(* Logix 5000 project; controller EIP_Test2 1769-L16ER-BB1B rev 21.11; software revision 21.00 *)

TASK MainTask (continuous, watchdog 500 ms) : MainProgram

MODULES
   Local : 1769-L16ER-BB1B (PointIO 0, rev 21.11)
      T2 : vendor 1316 type 43 code 256 (Ethernet 192.168.4.6, rev 2.86, StandardDataDriven RPI 10 ms)
      Laser : vendor 1316 type 43 code 256 (Ethernet 192.168.4.3, rev 2.86, StandardDataDriven RPI 10 ms)
      Discrete_IO : Embedded (PointIO 1, rev 21.11, Output RPI 20 ms)
END_MODULES

TYPE Job_Field :
STRUCT
   Field_Index : SINT;
   Uniqueness : SINT;
   Verify : SINT;
   Reserved : SINT;
END_STRUCT
END_TYPE

TYPE LEC_O2T :
STRUCT
   X_Offset_mm_x100 : INT;   // X axis offset in units of [millimeters times 100]
   Y_Offset_mm_x100 : INT;   // Y axis offset in units of [millimeters times 100]
   Rotation_deg_x10 : INT;   // Rotation in units of [degrees times 10]
   X_Rotation_Center_mm_x100 : INT;   // X coordinate of the center of rotation in units of [millimeters times 100]
   Y_Rotation_Center_mm_x100 : INT;   // Y coordinate of the center of rotation in units of [millimeters times 100]
   X_Scale_x1000 : INT;   // X scale factor in units of [scale times 1000]. For example, use 1000 for a scale of 1
   Y_Scale_x1000 : INT;   // Y scale factor in units of [scale times 1000]. For example, use 1000 for a scale of 1
   Reserved : INT;   // Reserved
   Marker_Command : INT;   // Numeric command from PLC to marker
   Computed_Job_Field_Index : INT;   // The field index number for the computed field
   Mark_Timeout_Sec : INT;   // The maximum time to allow for marking [seconds]. An error is generated if this time is exceeded.
   Reserved_1 : INT;   // Reserved
   Barcode_Pass_Grade : INT;   // Pass grade for barcode verification
   Max_Remarks : INT;   // Maximum number of remark attempts if camera verification fails
   Short_Job_Field : Job_Field[5];   // The field index numbers of up to five 32-character string fields
   Long_Job_Field : Job_Field;   // The field index numbers of a single 64-character string field
   Marker_Job_File_Name : String32;   // The name of the marker job file to load
   Camera_Job_File_Name : String32;   // The name of the camera job file to load
   Short_Field_String : String32[5];   // Short string field values [32-characters]
   Long_Field_String : String128;   // Long string field value [128-characters]
END_STRUCT
END_TYPE

TYPE LEC_T2O :
STRUCT
   Marker_State : INT;   // The numeric marker state
   Reserved : INT;
   Last_Mark_Cycle_Time_Ms : DINT;   // The elapsed cycle time, or cycle time of the last mark in milliseconds
   Status_Word : DINT;   // LEC Standard IO word
   Marker_Error_Code : INT;   // The marker error code (0 = No Error)
   Controller_Error_Code : INT;   // The controller error code (LEC or Couth) (0 = No Error)
   Heart_Beat : DINT;   // Heartbeat indicator. Increasing number.
   Input_Field_Checksum : DINT;   // Simple checksum of all input field bytes
   Echo_Job_File_Name : String32;   // An echo of the job file name that has been loaded
   Results_Field : String128;   // A string results field generated by the marker
   Marker_State_Desc : String64;   // A description of the current marker state
   Marker_Error_Desc : String128;   // A description of the current marker error
END_STRUCT
END_TYPE

TYPE MDrive_Inputs_T2O :
STRUCT
   BY : BOOL;
   MV : BOOL;
   IN : SINT;
   C1 : DINT;
   C2 : DINT;
   V : DINT;
END_STRUCT
END_TYPE

TYPE MDrive_Outputs_O2T :
STRUCT
   A : DINT;
   D : DINT;
   MA : DINT;
   MR : DINT;
   RC : SINT;
   HC : SINT;
   OT : SINT;
   SL : DINT;
   VI : DINT;
   VM : DINT;
   TE : SINT;
   D5 : SINT;
END_STRUCT
END_TYPE

TYPE String128 :
STRUCT
   LEN : DINT;
   DATA : SINT[128];
END_STRUCT
END_TYPE

TYPE String32 :
STRUCT
   LEN : DINT;
   DATA : SINT[32];
END_STRUCT
END_TYPE

TYPE String64 :
STRUCT
   LEN : DINT;
   DATA : SINT[64];
END_STRUCT
END_TYPE

ADD_ON_INSTRUCTION Acquire_Host_Mode   (* revision 1.0, vendor Mecco Marking & Traceability *)
VAR_IN_OUT
   Inputs : LEC_O2T; {required}
   Outputs : LEC_T2O; {required}
END_VAR
VAR_OUTPUT
   InProcess : BOOL; {access Read Only}
   Done : BOOL; {access Read Only}
END_VAR
VAR_IN_OUT
   nstate : DINT; {required}
END_VAR
VAR
   Comment : STRING; {access None}
END_VAR

ROUTINE Logic   (* ladder *)
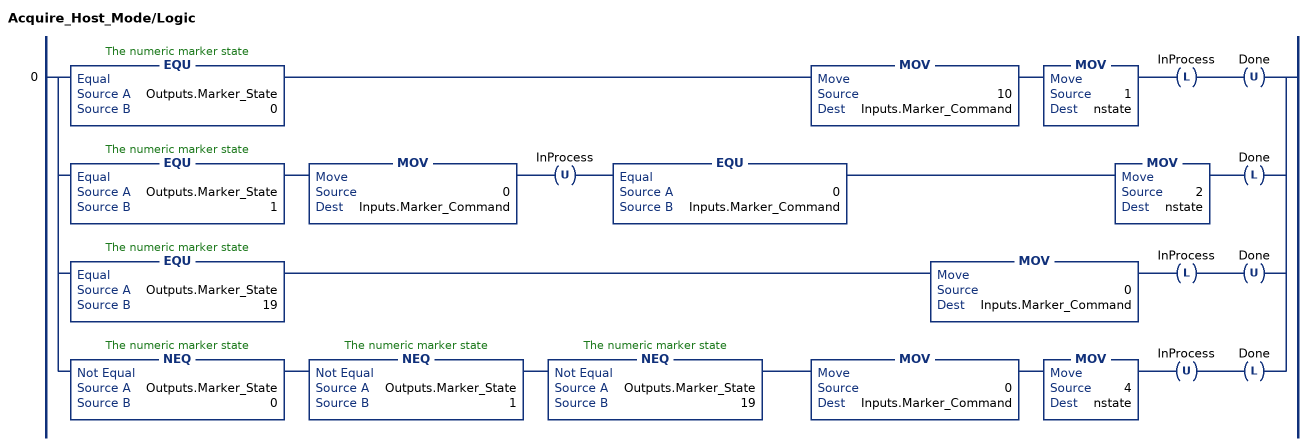
   0: [EQU(Outputs.Marker_State,0) MOV(10,Inputs.Marker_Command) MOV(1,nstate) OTL(InProcess) OTU(Done) ,EQU(Outputs.Marker_State,1) MOV(0,Inputs.Marker_Command) OTU(InProcess) EQU(0,Inputs.Marker_Command) MOV(2,nstate) OTL(Done) ,EQU(Outputs.Marker_State,19) MOV(0,Inputs.Marker_Command) OTL(InProcess) OTU(Done) ,NEQ(Outputs.Marker_State,0) NEQ(Outputs.Marker_State,1) NEQ(Outputs.Marker_State,19) MOV(0,Inputs.Marker_Command) MOV(4,nstate) OTU(InProcess) OTL(Done) ];
END_ROUTINE
END_ADD_ON_INSTRUCTION

ADD_ON_INSTRUCTION Clear_Error   (* revision 0.6, vendor Mecco Marking & Traceability *)
VAR_IN_OUT
   Inputs : LEC_O2T; {required}
   Outputs : LEC_T2O; {required}
END_VAR
VAR_OUTPUT
   Outcome : DINT; {access Read Only}
   InProcess : BOOL; {access Read Only}
   Done : BOOL; {access Read Only}
END_VAR
VAR_IN_OUT
   nstate : DINT; {required}
END_VAR
VAR
   Comment : STRING; {access None}
END_VAR

ROUTINE Logic   (* ladder *)
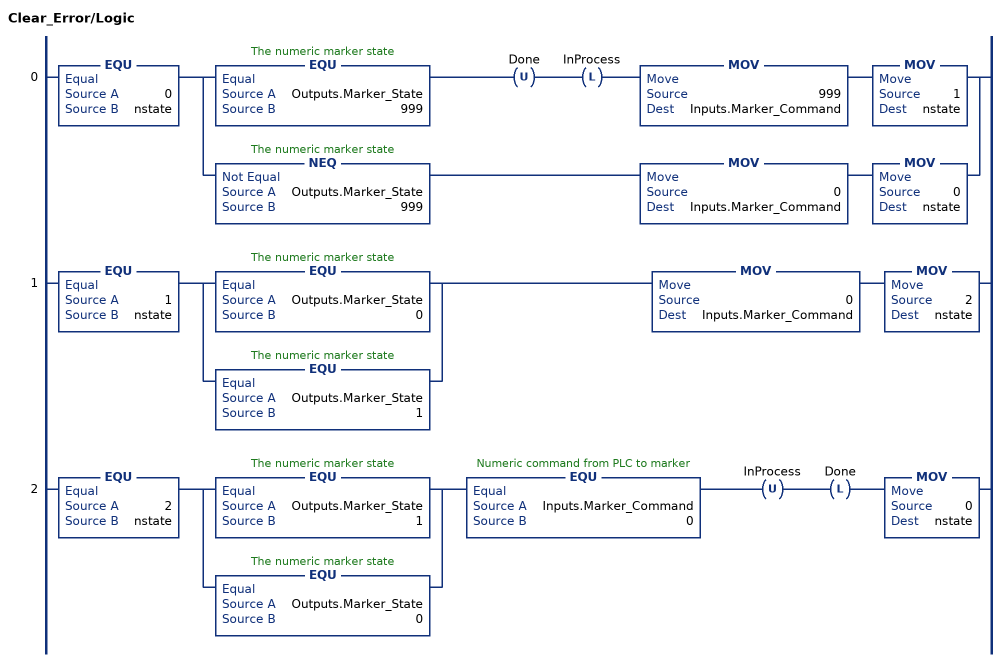
   0: EQU(0,nstate)[EQU(Outputs.Marker_State,999) OTU(Done) OTL(InProcess) MOV(999,Inputs.Marker_Command) MOV(1,nstate) ,NEQ(Outputs.Marker_State,999) MOV(0,Inputs.Marker_Command) MOV(0,nstate) ];
   1: EQU(1,nstate)[EQU(Outputs.Marker_State,0) ,EQU(Outputs.Marker_State,1) ]MOV(0,Inputs.Marker_Command)MOV(2,nstate);
   2: EQU(2,nstate)[EQU(Outputs.Marker_State,1) ,EQU(Outputs.Marker_State,0) ]EQU(Inputs.Marker_Command,0)OTU(InProcess)OTL(Done)MOV(0,nstate);
END_ROUTINE
END_ADD_ON_INSTRUCTION

ADD_ON_INSTRUCTION Load_Job   (* revision 1.0, vendor Mecco Marking & Traceability *)
VAR_IN_OUT
   Inputs : LEC_O2T; {required}
   Outputs : LEC_T2O; {required}
END_VAR
VAR_OUTPUT
   InProcess : BOOL; {access Read Only}
   Done : BOOL; {access Read Only}
END_VAR
VAR_IN_OUT
   Job_File_Name : STRING; {required}
END_VAR
VAR_OUTPUT
   Error : BOOL; {access Read Only}
END_VAR
VAR_INPUT
   Reset : BOOL;
END_VAR
VAR_IN_OUT
   nstate : DINT; {required}
END_VAR
VAR
   Comment : STRING; {access None}
   ErrorTimer : TIMER := (PRE := 5000); {access None}
   State1ONS : BOOL; {access None}
   BLANKSTRING : STRING; {access None}
   tnstate2 : TIMER := (PRE := 4000); {access None}
END_VAR

ROUTINE Logic   (* ladder *)
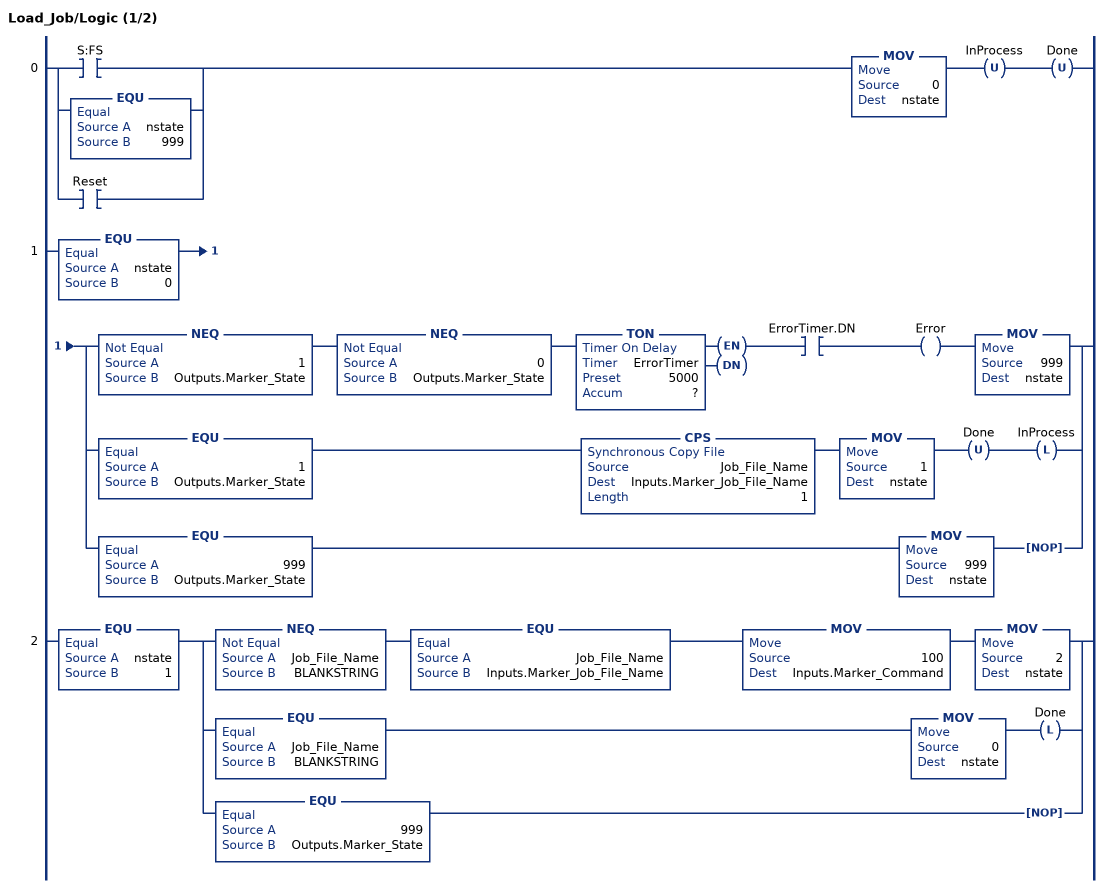
   0: [XIC(S:FS) ,EQU(nstate,999) ,XIC(Reset) ]MOV(0,nstate)OTU(InProcess)OTU(Done);
   1: EQU(nstate,0)[[NEQ(1,Outputs.Marker_State) NEQ(0,Outputs.Marker_State) TON(ErrorTimer,?,?) XIC(ErrorTimer.DN) OTE(Error) MOV(999,nstate) ,EQU(1,Outputs.Marker_State) CPS(Job_File_Name,Inputs.Marker_Job_File_Name,1) MOV(1,nstate) OTU(Done) OTL(InProcess) ] ,EQU(999,Outputs.Marker_State) MOV(999,nstate) NOP() ];
   2: EQU(nstate,1)[NEQ(Job_File_Name,BLANKSTRING) EQU(Job_File_Name,Inputs.Marker_Job_File_Name) MOV(100,Inputs.Marker_Command) MOV(2,nstate) ,EQU(Job_File_Name,BLANKSTRING) MOV(0,nstate) OTL(Done) ,EQU(999,Outputs.Marker_State) NOP() ];
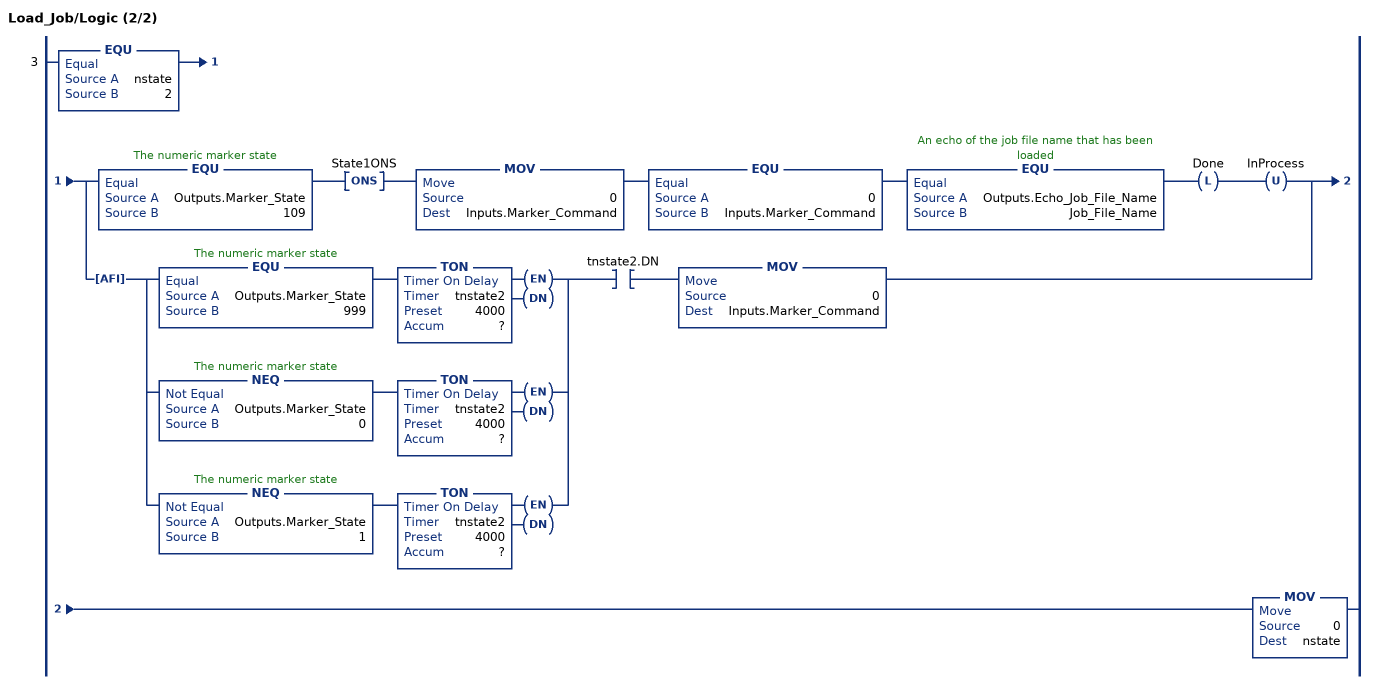
   3: EQU(nstate,2)[EQU(Outputs.Marker_State,109) ONS(State1ONS) MOV(0,Inputs.Marker_Command) EQU(0,Inputs.Marker_Command) EQU(Outputs.Echo_Job_File_Name,Job_File_Name) OTL(Done) OTU(InProcess) ,AFI() [EQU(Outputs.Marker_State,999) TON(tnstate2,?,?) ,NEQ(Outputs.Marker_State,0) TON(tnstate2,?,?) ,NEQ(Outputs.Marker_State,1) TON(tnstate2,?,?) ] XIC(tnstate2.DN) MOV(0,Inputs.Marker_Command) ]MOV(0,nstate);
END_ROUTINE
END_ADD_ON_INSTRUCTION

ADD_ON_INSTRUCTION Load_Job_T2   (* revision 1.0, vendor Mecco Marking & Traceability *)
VAR_IN_OUT
   Inputs : LEC_O2T; {required}
   Outputs : LEC_T2O; {required}
END_VAR
VAR_OUTPUT
   InProcess : BOOL; {access Read Only}
   Done : BOOL; {access Read Only}
END_VAR
VAR_IN_OUT
   Job_File_Name : STRING; {required}
END_VAR
VAR_OUTPUT
   Error : BOOL; {access Read Only}
END_VAR
VAR_INPUT
   Reset : BOOL;
END_VAR
VAR
   Comment : STRING; {access None}
   ErrorTimer : TIMER := (PRE := 5000); {access None}
   State1ONS : BOOL; {access None}
   BLANKSTRING : STRING; {access None}
   nstate : DINT; {access None}
END_VAR

ROUTINE Logic   (* ladder *)
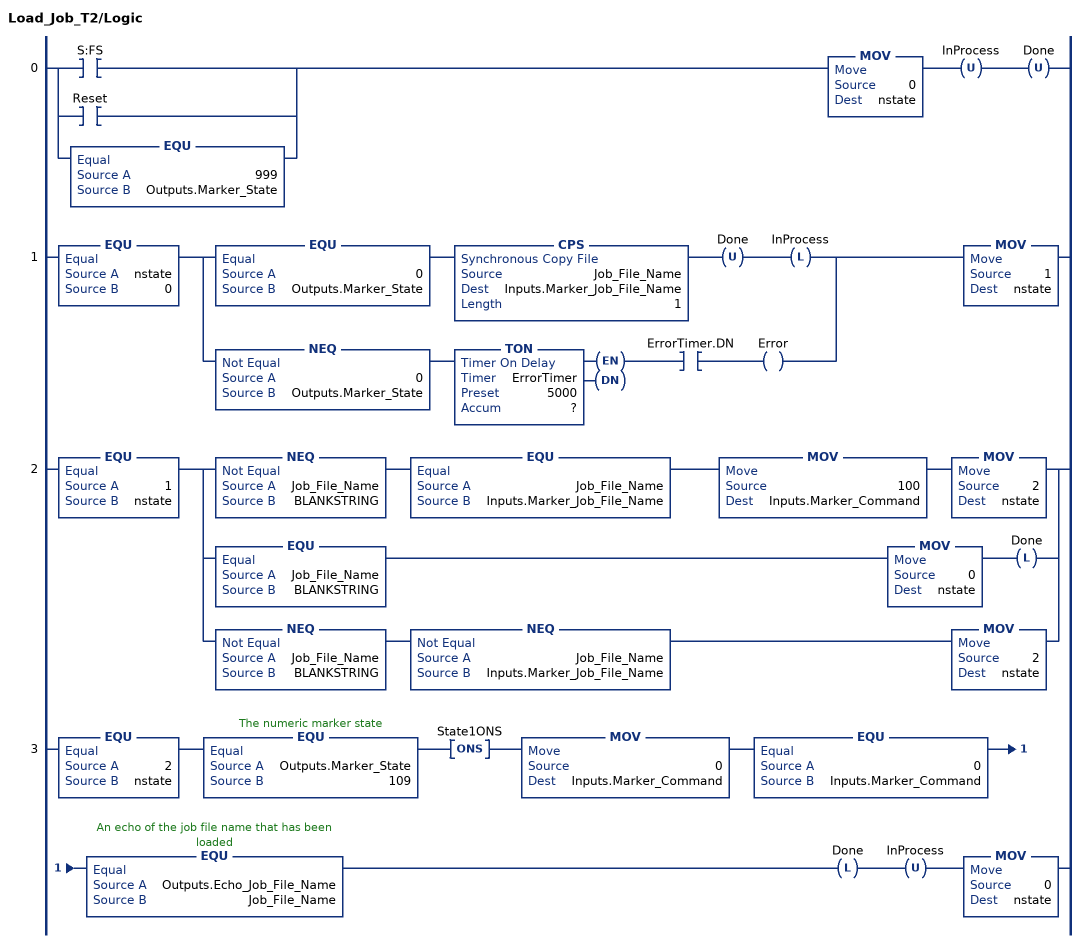
   0: [XIC(S:FS) ,XIC(Reset) ,EQU(999,Outputs.Marker_State) ]MOV(0,nstate)OTU(InProcess)OTU(Done);
   1: EQU(nstate,0)[EQU(0,Outputs.Marker_State) CPS(Job_File_Name,Inputs.Marker_Job_File_Name,1) OTU(Done) OTL(InProcess) ,NEQ(0,Outputs.Marker_State) TON(ErrorTimer,?,?) XIC(ErrorTimer.DN) OTE(Error) ]MOV(1,nstate);
   2: EQU(1,nstate)[NEQ(Job_File_Name,BLANKSTRING) EQU(Job_File_Name,Inputs.Marker_Job_File_Name) MOV(100,Inputs.Marker_Command) MOV(2,nstate) ,EQU(Job_File_Name,BLANKSTRING) MOV(0,nstate) OTL(Done) ,NEQ(Job_File_Name,BLANKSTRING) NEQ(Job_File_Name,Inputs.Marker_Job_File_Name) MOV(2,nstate) ];
   3: EQU(2,nstate)EQU(Outputs.Marker_State,109)ONS(State1ONS)MOV(0,Inputs.Marker_Command)EQU(0,Inputs.Marker_Command)EQU(Outputs.Echo_Job_File_Name,Job_File_Name)OTL(Done)OTU(InProcess)MOV(0,nstate);
END_ROUTINE
END_ADD_ON_INSTRUCTION

ADD_ON_INSTRUCTION Load_Variables   (* revision 1.0, vendor Mecco Marking & Traceability *)
VAR_IN_OUT
   Inputs : LEC_O2T; {required}
   Outputs : LEC_T2O; {required}
END_VAR
VAR_OUTPUT
   InProcess : BOOL; {access Read Only}
   Done : BOOL; {access Read Only}
END_VAR
VAR_IN_OUT
   Short_Variable_1_Text : STRING; {required}
END_VAR
VAR_INPUT
   Short_Variable_1_ObjectNum : DINT; {access None}
END_VAR
VAR_IN_OUT
   Short_Variable_2_Text : STRING; {required}
END_VAR
VAR_INPUT
   Short_Variable_2_ObjectNum : DINT; {access None}
END_VAR
VAR_IN_OUT
   Short_Variable_3_Text : STRING; {required}
END_VAR
VAR_INPUT
   Short_Variable_3_ObjectNum : DINT; {access None}
END_VAR
VAR_IN_OUT
   Short_Variable_4_Text : STRING; {required}
END_VAR
VAR_INPUT
   Short_Variable_4_ObjectNum : DINT; {access None}
END_VAR
VAR_IN_OUT
   Short_Variable_5_Text : STRING; {required}
END_VAR
VAR_INPUT
   Short_Variable_5_ObjectNum : DINT; {access None}
END_VAR
VAR_IN_OUT
   Long_Variable_Text : STRING; {required}
END_VAR
VAR_INPUT
   Long_Variable_ObjectNum : DINT; {access None}
END_VAR
VAR
   Comment : STRING; {access None}
   nstate : DINT := 3; {access None}
END_VAR

ROUTINE Logic   (* ladder *)
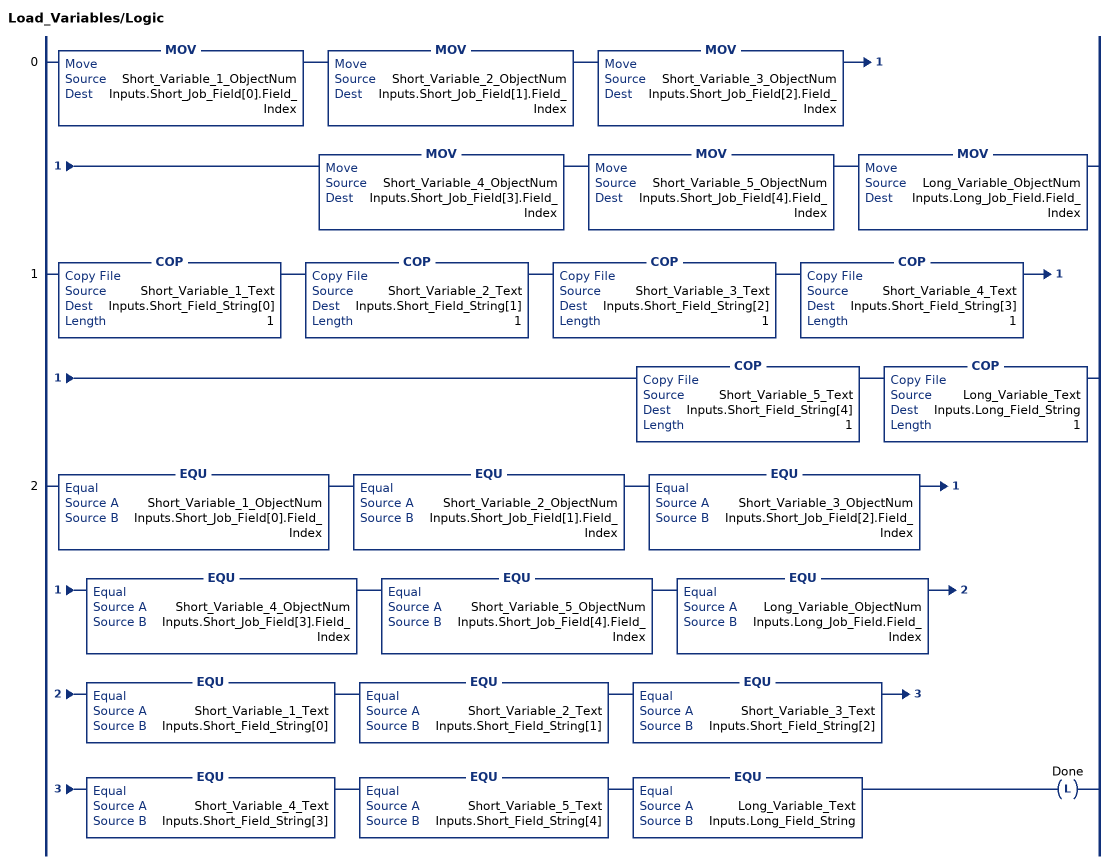
   0: MOV(Short_Variable_1_ObjectNum,Inputs.Short_Job_Field[0].Field_Index)MOV(Short_Variable_2_ObjectNum,Inputs.Short_Job_Field[1].Field_Index)MOV(Short_Variable_3_ObjectNum,Inputs.Short_Job_Field[2].Field_Index)MOV(Short_Variable_4_ObjectNum,Inputs.Short_Job_Field[3].Field_Index)MOV(Short_Variable_5_ObjectNum,Inputs.Short_Job_Field[4].Field_Index)MOV(Long_Variable_ObjectNum,Inputs.Long_Job_Field.Field_Index);
   1: COP(Short_Variable_1_Text,Inputs.Short_Field_String[0],1)COP(Short_Variable_2_Text,Inputs.Short_Field_String[1],1)COP(Short_Variable_3_Text,Inputs.Short_Field_String[2],1)COP(Short_Variable_4_Text,Inputs.Short_Field_String[3],1)COP(Short_Variable_5_Text,Inputs.Short_Field_String[4],1)COP(Long_Variable_Text,Inputs.Long_Field_String,1);
   2: EQU(Short_Variable_1_ObjectNum,Inputs.Short_Job_Field[0].Field_Index)EQU(Short_Variable_2_ObjectNum,Inputs.Short_Job_Field[1].Field_Index)EQU(Short_Variable_3_ObjectNum,Inputs.Short_Job_Field[2].Field_Index)EQU(Short_Variable_4_ObjectNum,Inputs.Short_Job_Field[3].Field_Index)EQU(Short_Variable_5_ObjectNum,Inputs.Short_Job_Field[4].Field_Index)EQU(Long_Variable_ObjectNum,Inputs.Long_Job_Field.Field_Index)EQU(Short_Variable_1_Text,Inputs.Short_Field_String[0])EQU(Short_Variable_2_Text,Inputs.Short_Field_String[1])EQU(Short_Variable_3_Text,Inputs.Short_Field_String[2])EQU(Short_Variable_4_Text,Inputs.Short_Field_String[3])EQU(Short_Variable_5_Text,Inputs.Short_Field_String[4])EQU(Long_Variable_Text,Inputs.Long_Field_String)OTL(Done);
END_ROUTINE
END_ADD_ON_INSTRUCTION

ADD_ON_INSTRUCTION Mark_Job   (* revision 1.0, vendor Mecco Marking & Traceability *)
VAR_IN_OUT
   Inputs : LEC_O2T; {required}
   Outputs : LEC_T2O; {required}
END_VAR
VAR_OUTPUT
   InProcess : BOOL; {access Read Only}
   Done : BOOL; {access Read Only}
   Error : BOOL; {access Read Only}
   MarkInProgress : BOOL; {access Read Only, visible}
END_VAR
VAR_INPUT
   Reset : BOOL;
END_VAR
VAR_IN_OUT
   nstate : DINT; {required}
END_VAR
VAR
   Comment : STRING; {access None}
   ErrorTimer : TIMER := (PRE := 5000); {access None}
END_VAR

ROUTINE Logic   (* ladder *)
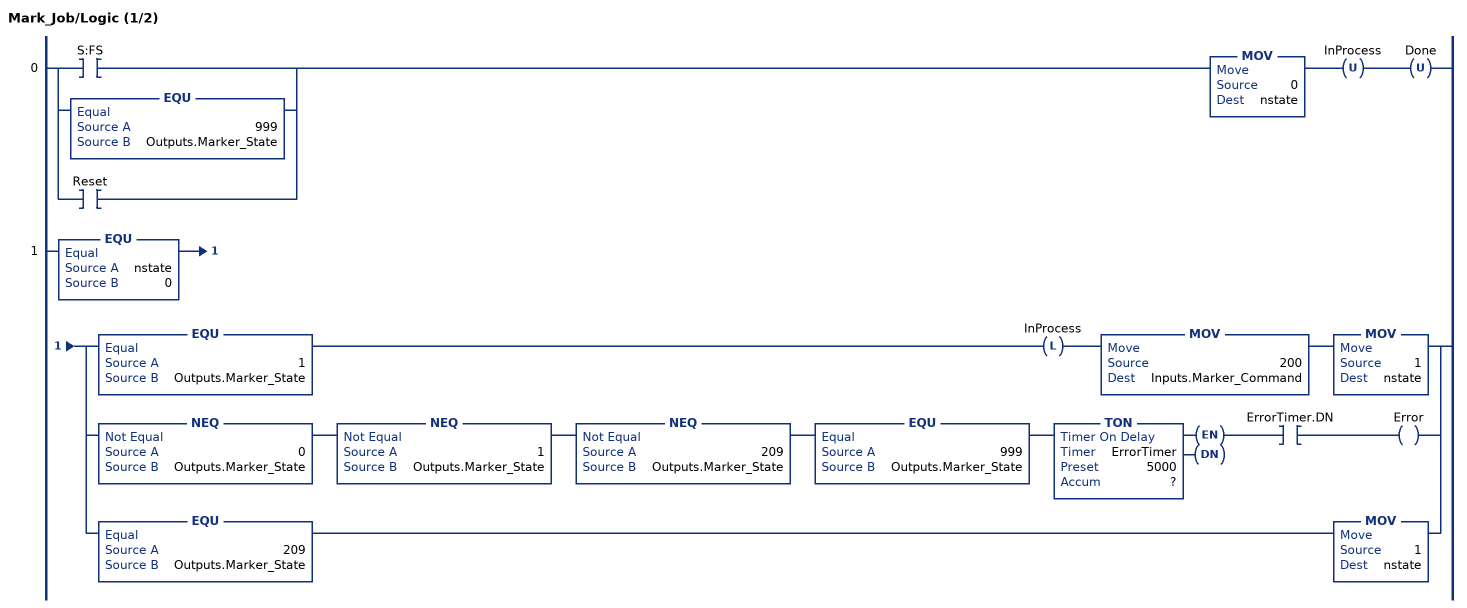
   0: [XIC(S:FS) ,EQU(999,Outputs.Marker_State) ,XIC(Reset) ]MOV(0,nstate)OTU(InProcess)OTU(Done);
   1: EQU(nstate,0)[EQU(1,Outputs.Marker_State) OTL(InProcess) MOV(200,Inputs.Marker_Command) MOV(1,nstate) ,NEQ(0,Outputs.Marker_State) NEQ(1,Outputs.Marker_State) NEQ(209,Outputs.Marker_State) EQU(999,Outputs.Marker_State) TON(ErrorTimer,?,?) XIC(ErrorTimer.DN) OTE(Error) ,EQU(209,Outputs.Marker_State) MOV(1,nstate) ];
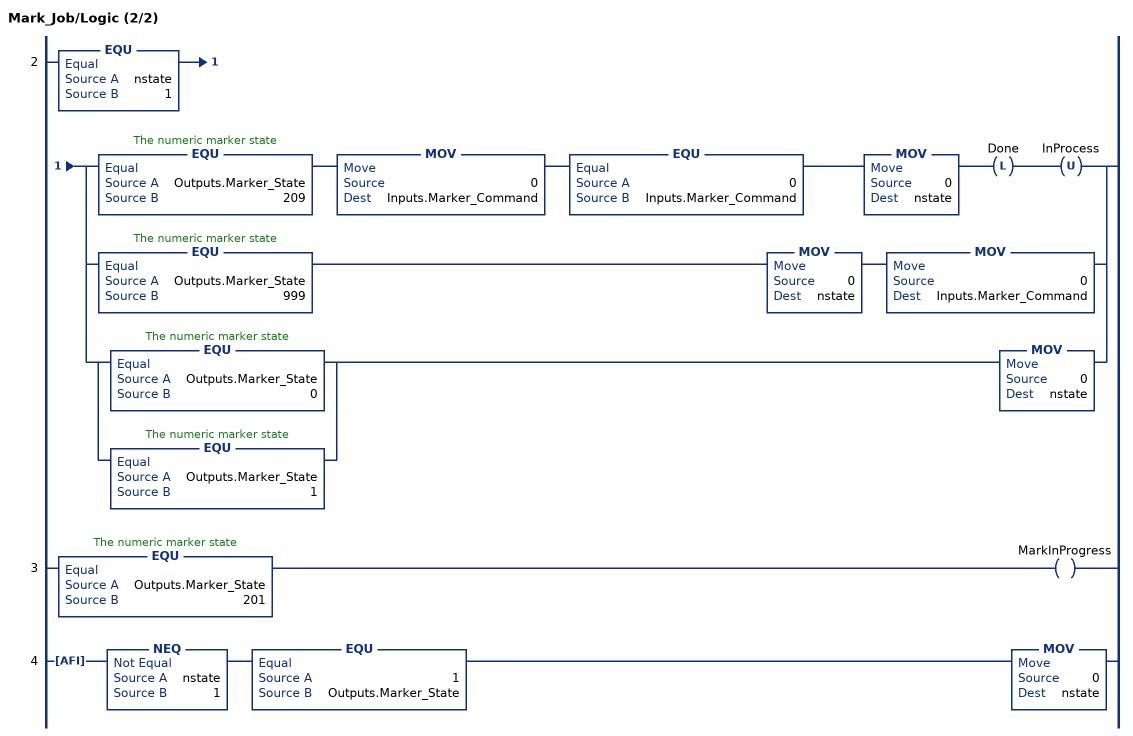
   2: EQU(nstate,1)[EQU(Outputs.Marker_State,209) MOV(0,Inputs.Marker_Command) EQU(0,Inputs.Marker_Command) MOV(0,nstate) OTL(Done) OTU(InProcess) ,EQU(Outputs.Marker_State,999) MOV(0,nstate) MOV(0,Inputs.Marker_Command) ,[EQU(Outputs.Marker_State,0) ,EQU(Outputs.Marker_State,1) ] MOV(0,nstate) ];
   3: EQU(Outputs.Marker_State,201)OTE(MarkInProgress);
   4: AFI()NEQ(nstate,1)EQU(1,Outputs.Marker_State)MOV(0,nstate);
END_ROUTINE
END_ADD_ON_INSTRUCTION

ADD_ON_INSTRUCTION Mark_Job_T2   (* revision 1.0, vendor Mecco Marking & Traceability *)
VAR_IN_OUT
   Inputs : LEC_O2T; {required}
   Outputs : LEC_T2O; {required}
END_VAR
VAR_OUTPUT
   InProcess : BOOL; {access Read Only}
   Done : BOOL; {access Read Only}
   Error : BOOL; {access Read Only}
   MarkInProgress : BOOL; {access Read Only, visible}
END_VAR
VAR_INPUT
   Reset : BOOL;
END_VAR
VAR
   Comment : STRING; {access None}
   ErrorTimer : TIMER := (PRE := 5000); {access None}
   nstate : DINT; {access None}
END_VAR

ROUTINE Logic   (* ladder *)
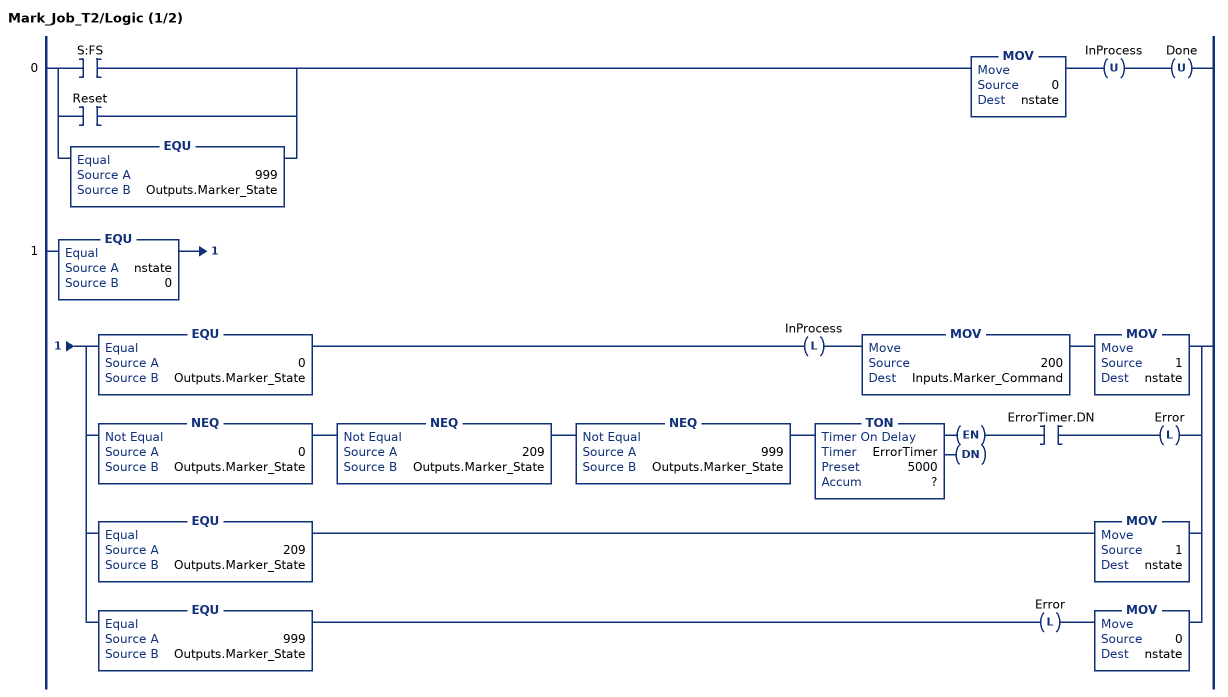
   0: [XIC(S:FS) ,[XIC(Reset) ,EQU(999,Outputs.Marker_State) ] ]MOV(0,nstate)OTU(InProcess)OTU(Done);
   1: EQU(nstate,0)[EQU(0,Outputs.Marker_State) OTL(InProcess) MOV(200,Inputs.Marker_Command) MOV(1,nstate) ,NEQ(0,Outputs.Marker_State) NEQ(209,Outputs.Marker_State) NEQ(999,Outputs.Marker_State) TON(ErrorTimer,?,?) XIC(ErrorTimer.DN) OTL(Error) ,EQU(209,Outputs.Marker_State) MOV(1,nstate) ,EQU(999,Outputs.Marker_State) OTL(Error) MOV(0,nstate) ];
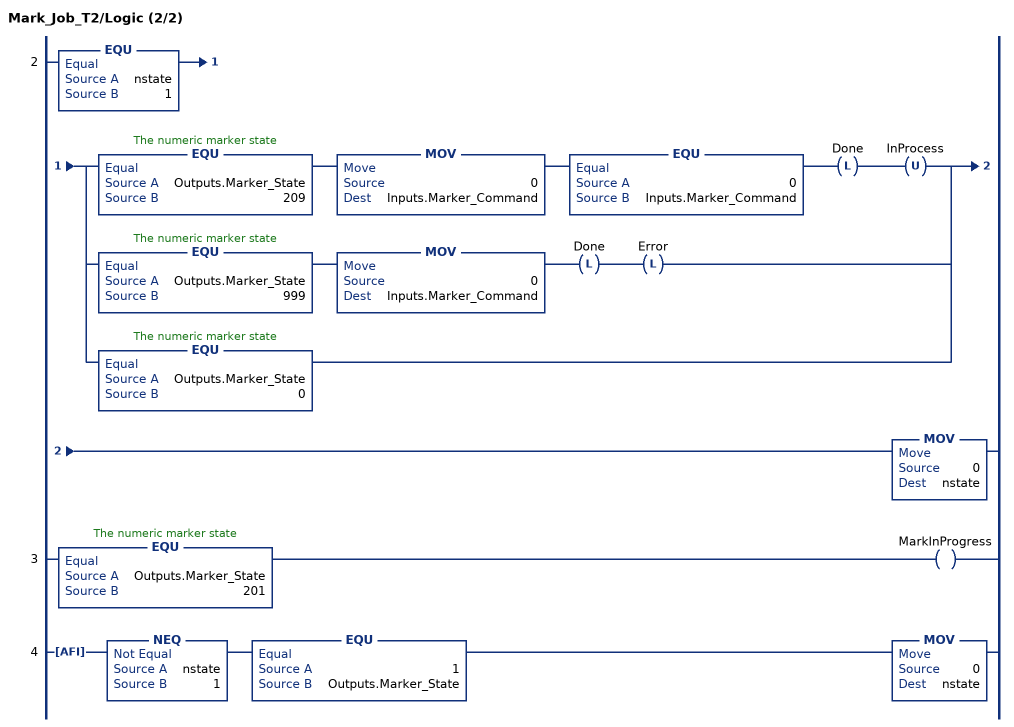
   2: EQU(nstate,1)[EQU(Outputs.Marker_State,209) MOV(0,Inputs.Marker_Command) EQU(0,Inputs.Marker_Command) OTL(Done) OTU(InProcess) ,EQU(Outputs.Marker_State,999) MOV(0,Inputs.Marker_Command) OTL(Done) OTL(Error) ,EQU(Outputs.Marker_State,0) ]MOV(0,nstate);
   3: EQU(Outputs.Marker_State,201)OTE(MarkInProgress);
   4: AFI()NEQ(nstate,1)EQU(1,Outputs.Marker_State)MOV(0,nstate);
END_ROUTINE
END_ADD_ON_INSTRUCTION

ADD_ON_INSTRUCTION Release_Host_Mode   (* revision 1.0, vendor Mecco Marking & Traceability *)
VAR_IN_OUT
   Inputs : LEC_O2T; {required}
   Outputs : LEC_T2O; {required}
END_VAR
VAR_OUTPUT
   InProcess : BOOL; {access Read Only}
   Done : BOOL; {access Read Only}
END_VAR
VAR
   Comment : STRING; {access None}
   nstate : DINT; {access None}
END_VAR

ROUTINE Logic   (* ladder *)
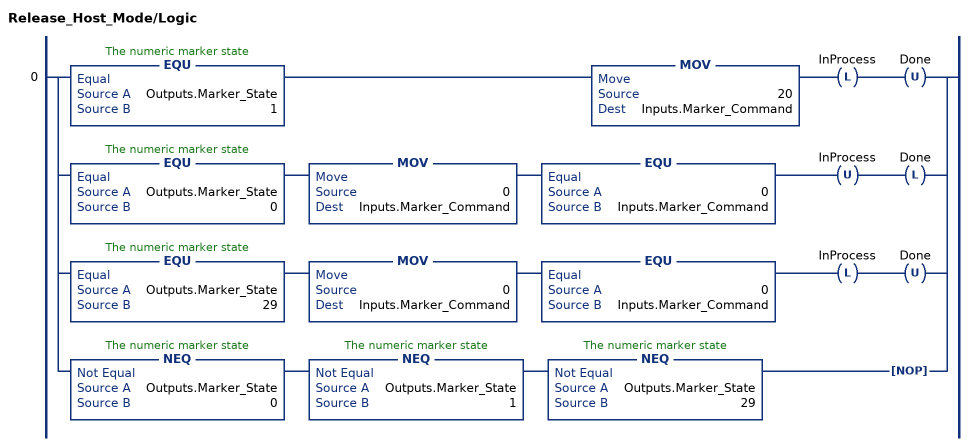
   0: [EQU(Outputs.Marker_State,1) MOV(20,Inputs.Marker_Command) OTL(InProcess) OTU(Done) ,EQU(Outputs.Marker_State,0) MOV(0,Inputs.Marker_Command) EQU(0,Inputs.Marker_Command) OTU(InProcess) OTL(Done) ,EQU(Outputs.Marker_State,29) MOV(0,Inputs.Marker_Command) EQU(0,Inputs.Marker_Command) OTL(InProcess) OTU(Done) ,NEQ(Outputs.Marker_State,0) NEQ(Outputs.Marker_State,1) NEQ(Outputs.Marker_State,29) NOP() ];
END_ROUTINE
END_ADD_ON_INSTRUCTION

VAR_GLOBAL   (* controller tags *)
   AcquireHost_nState : DINT;
   AOI_Acquire_Host_Laser : Acquire_Host_Mode;
   AOI_Load_Job : Load_Job;
   AOI_Load_Job_T2 : Load_Job_T2;
   AOI_Load_Variables : Load_Variables;
   AOI_Load_Variables_T2 : Load_Variables;
   AOI_Mark_Job : Mark_Job;
   AOI_Mark_Job_T2 : Mark_Job_T2;
   AOI_Release_Host : Release_Host_Mode;
   Dot_Peen_Input : LEC_O2T := (X_Scale_x1000 := 1000, Y_Scale_x1000 := 1000, Mark_Timeout_Sec := 999, Short_Job_Field[0].Field_Index := 1, Short_Job_Field[1].Field_Index := 2, Short_Job_Field[2].Field_Index := 3, Short_Job_Field[3].Field_Index := 4, Short_Job_Field[4].Field_Index := 5, Marker_Job_File_Name := 'Test1000.txt', Short_Field_String[0] := 'Line1', Short_Field_String[1] := 'Line2', Short_Field_String[2] := 'Line3', Short_Field_String[3] := 'Line4', Short_Field_String[4] := 'Line5');
   Dot_Peen_Load_Job : BOOL;
   Dot_Peen_Load_Variables : BOOL;
   Dot_Peen_Mark_Job : BOOL;
   Dot_Peen_Output : LEC_T2O := (Last_Mark_Cycle_Time_Ms := 4945, Heart_Beat := 345199, Input_Field_Checksum := 3222, Echo_Job_File_Name := 'Test1000.txt', Marker_State_Desc := '[1] Ready', Marker_Error_Desc := 'No error');
   HMI_Bits : DINT := 1;
   Job : BOOL;
   Laser_Acquire : BOOL;
   Laser_Acquire_Host : BOOL;
   Laser_Inputs : LEC_O2T := (X_Scale_x1000 := 1000, Y_Scale_x1000 := 1000, Mark_Timeout_Sec := 999, Short_Job_Field[0].Field_Index := 1, Short_Job_Field[1].Field_Index := 2, Short_Job_Field[2].Field_Index := 3, Short_Job_Field[3].Field_Index := 4, Short_Job_Field[4].Field_Index := 5, Marker_Job_File_Name := 'TAG1.DAT', Short_Field_String[0] := 'Line1', Short_Field_String[1] := 'Line2', Short_Field_String[2] := 'Line3', Short_Field_String[3] := 'Line4', Short_Field_String[4] := 'Line5', Long_Field_String := '590.00,3537,500,300,30,204.000,150,75,0,40.00,2.0,0,0,0,0,0.0,1,0,2.550,2.550,0.0,0.0,0,0');
   Laser_JobFileName : STRING;
   Laser_Load_Job : BOOL;
   Laser_Load_Variables : BOOL;
   Laser_Mark_Job : BOOL;
   Laser_Online_String : STRING := 'Ready to Fire';
   Laser_Outputs : LEC_T2O := (Marker_State := 1, Heart_Beat := 516904, Input_Field_Checksum := 7119, Echo_Job_File_Name := 'TAG1.DAT', Results_Field := '1405', Marker_State_Desc := '[1] Ready: Host Mode active', Marker_Error_Desc := 'No error');
   Laser_Release_Host : BOOL;
   LoadJob_nState : DINT;
   Long : STRING;
   Long_T2 : STRING;
   MarkJob_nState : DINT;
   MDive_Inputs : MDrive_Inputs_T2O;
   MDrive_Outputs : MDrive_Outputs_O2T;
   Short : STRING[5];
   Short_T2 : STRING[5];
   T2_JobFileName : STRING;
END_VAR

PROGRAM MainProgram   (* main routine MainRoutine *)
VAR
   B_Reset_Marker : BOOL;
   bDotPeenEnabled : BOOL := 1;
   Blank_String : String32;
   bLaserEnabled : BOOL := 1;
   bPauseDotPeen : BOOL;
   bPauseLaser : BOOL;
   Dot_Peen_Job_File_Name : String32 := 'Test1000.txt';
   Dot_Peen_Run_Counter : COUNTER := (ACC := 12, DN := 1);
   Dot_Peen_Start_Button : BOOL := 1;
   Field : String32[5] := ([0] := 'Line1', [1] := 'Line2', [2] := 'Line3', [3] := 'Line4', [4] := 'Line5');
   Job_File_Name : STRING := 'Series0_Text.dat';
   l_hstate : DINT;
   l_on : TIMER := (PRE := 12000);
   Laser_Heartbeat_Old : DINT := 1306452;
   Laser_Run_Counter : COUNTER := (ACC := 5, CU := 1, DN := 1);
   LASER_RUNNING : BOOL;
   LEC_Latch : BOOL;
   lHeartbeat_Check : BOOL := 1;
   lheartbeat_Timer : TIMER := (PRE := 1000);
   M_Drive_Accel_1 : BOOL;
   M_Drive_Decel_1 : BOOL;
   M_Drive_Position_1 : BOOL;
   M_Drive_Query_SN : BOOL;
   M_Drive_Reverse_1 : BOOL;
   M_Drive_Slew_1 : BOOL;
   M_Drive_Stop : BOOL;
   M_Drive_Velocity_1 : BOOL;
   MDrive_Out : DINT;
   nState : DINT;
   nState_DotPeen : DINT;
   Reset_Dot_Peen_Counter : BOOL;
   Reset_Laser_Counter : BOOL;
   Start_Button : BOOL := 1;
   T2_Latch : BOOL := 1;
   T_MarkerResetTimer : TIMER;
END_VAR

ROUTINE Dot_Peen   (* ladder *)
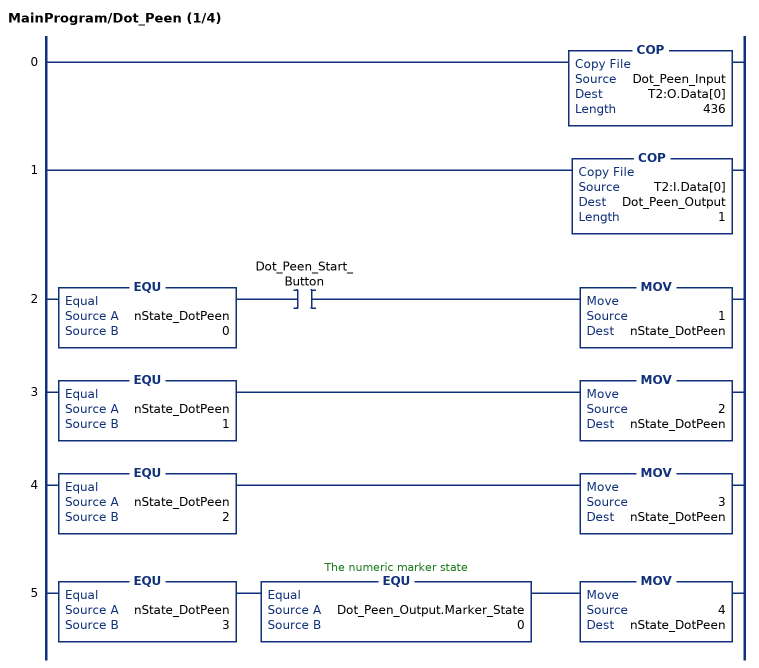
   0: COP(Dot_Peen_Input,T2:O.Data[0],436);
   1: COP(T2:I.Data[0],Dot_Peen_Output,1);
   2: EQU(nState_DotPeen,0)XIC(Dot_Peen_Start_Button)MOV(1,nState_DotPeen);
   3: EQU(nState_DotPeen,1)MOV(2,nState_DotPeen);
   4: EQU(nState_DotPeen,2)MOV(3,nState_DotPeen);
   5: EQU(nState_DotPeen,3)EQU(Dot_Peen_Output.Marker_State,0)MOV(4,nState_DotPeen);
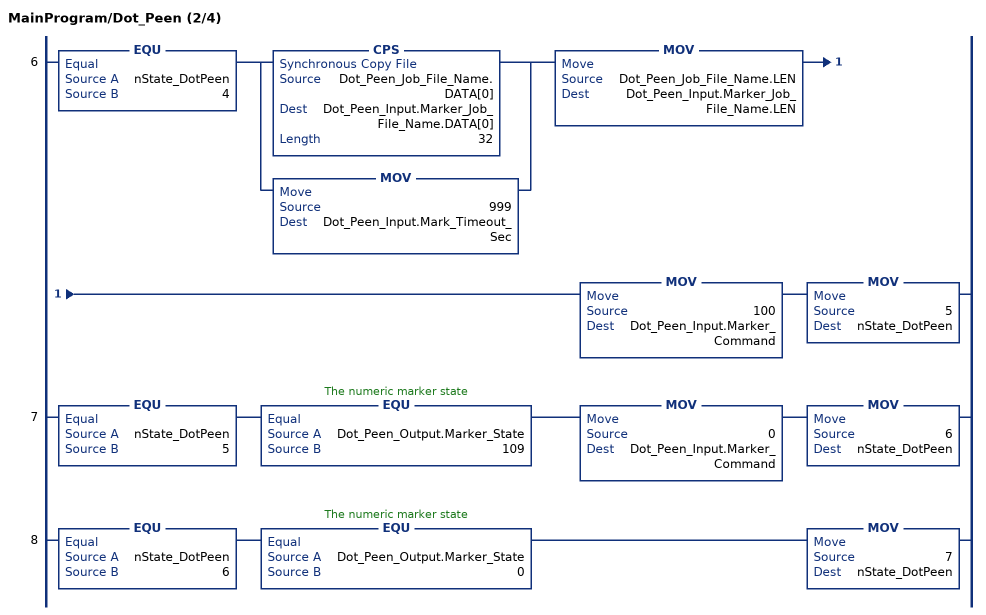
   6: EQU(nState_DotPeen,4)[CPS(Dot_Peen_Job_File_Name.DATA[0],Dot_Peen_Input.Marker_Job_File_Name.DATA[0],32) ,MOV(999,Dot_Peen_Input.Mark_Timeout_Sec) ]MOV(Dot_Peen_Job_File_Name.LEN,Dot_Peen_Input.Marker_Job_File_Name.LEN)MOV(100,Dot_Peen_Input.Marker_Command)MOV(5,nState_DotPeen);
   7: EQU(nState_DotPeen,5)EQU(Dot_Peen_Output.Marker_State,109)MOV(0,Dot_Peen_Input.Marker_Command)MOV(6,nState_DotPeen);
   8: EQU(nState_DotPeen,6)EQU(Dot_Peen_Output.Marker_State,0)MOV(7,nState_DotPeen);
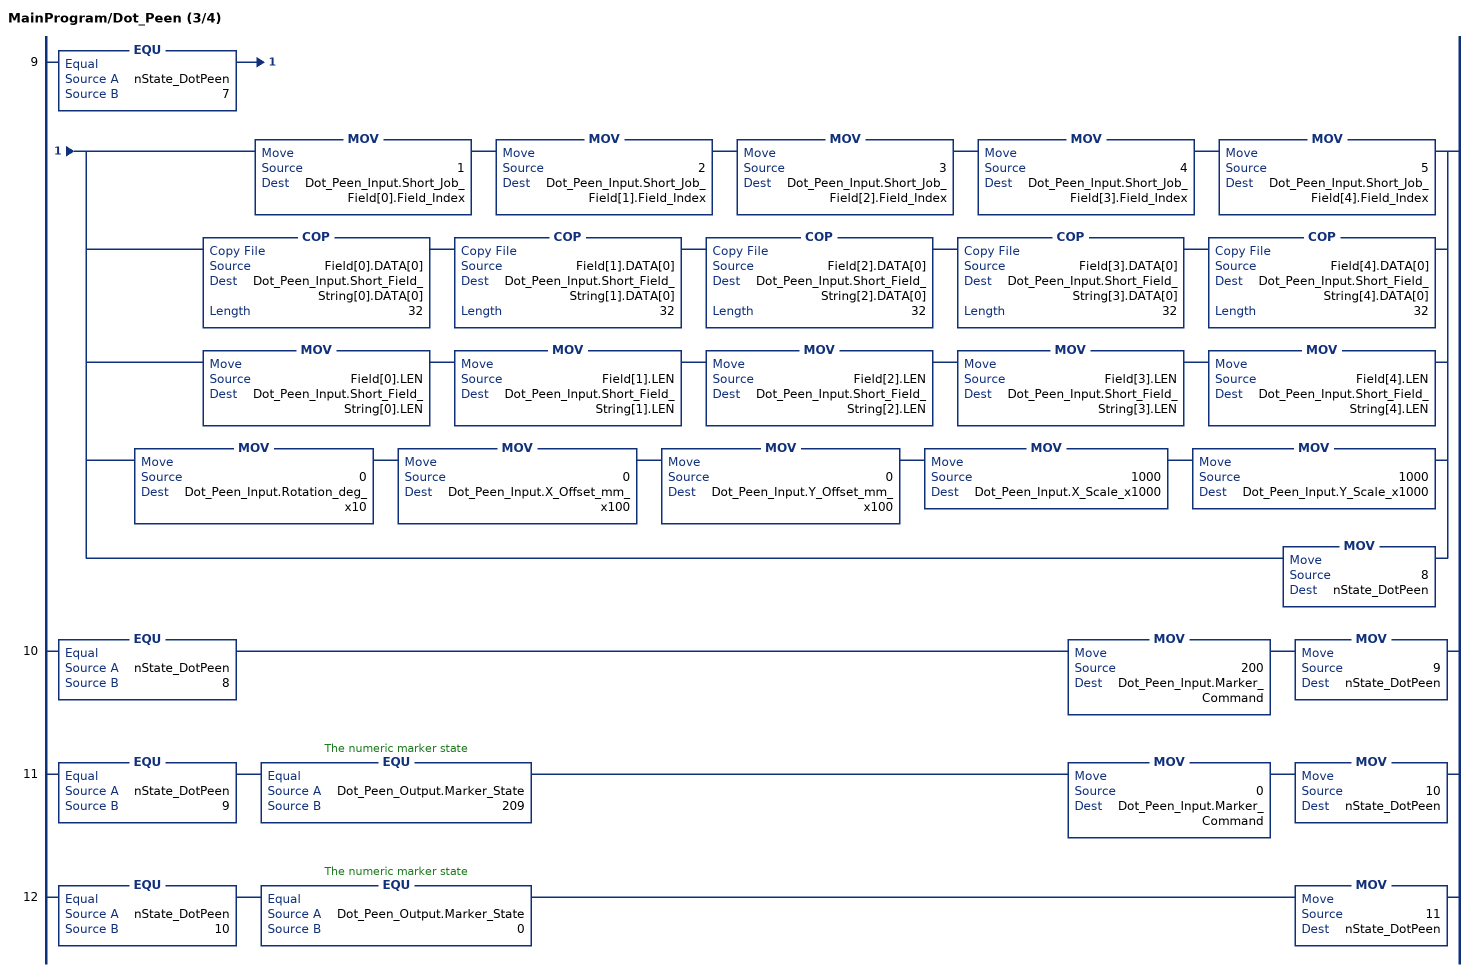
   9: EQU(nState_DotPeen,7)[MOV(1,Dot_Peen_Input.Short_Job_Field[0].Field_Index) MOV(2,Dot_Peen_Input.Short_Job_Field[1].Field_Index) MOV(3,Dot_Peen_Input.Short_Job_Field[2].Field_Index) MOV(4,Dot_Peen_Input.Short_Job_Field[3].Field_Index) MOV(5,Dot_Peen_Input.Short_Job_Field[4].Field_Index) ,COP(Field[0].DATA[0],Dot_Peen_Input.Short_Field_String[0].DATA[0],32) COP(Field[1].DATA[0],Dot_Peen_Input.Short_Field_String[1].DATA[0],32) COP(Field[2].DATA[0],Dot_Peen_Input.Short_Field_String[2].DATA[0],32) COP(Field[3].DATA[0],Dot_Peen_Input.Short_Field_String[3].DATA[0],32) COP(Field[4].DATA[0],Dot_Peen_Input.Short_Field_String[4].DATA[0],32) ,MOV(Field[0].LEN,Dot_Peen_Input.Short_Field_String[0].LEN) MOV(Field[1].LEN,Dot_Peen_Input.Short_Field_String[1].LEN) MOV(Field[2].LEN,Dot_Peen_Input.Short_Field_String[2].LEN) MOV(Field[3].LEN,Dot_Peen_Input.Short_Field_String[3].LEN) MOV(Field[4].LEN,Dot_Peen_Input.Short_Field_String[4].LEN) ,MOV(0,Dot_Peen_Input.Rotation_deg_x10) MOV(0,Dot_Peen_Input.X_Offset_mm_x100) MOV(0,Dot_Peen_Input.Y_Offset_mm_x100) MOV(1000,Dot_Peen_Input.X_Scale_x1000) MOV(1000,Dot_Peen_Input.Y_Scale_x1000) ,MOV(8,nState_DotPeen) ];
   10: EQU(nState_DotPeen,8)MOV(200,Dot_Peen_Input.Marker_Command)MOV(9,nState_DotPeen);
   11: EQU(nState_DotPeen,9)EQU(Dot_Peen_Output.Marker_State,209)MOV(0,Dot_Peen_Input.Marker_Command)MOV(10,nState_DotPeen);
   12: EQU(nState_DotPeen,10)EQU(Dot_Peen_Output.Marker_State,0)MOV(11,nState_DotPeen);
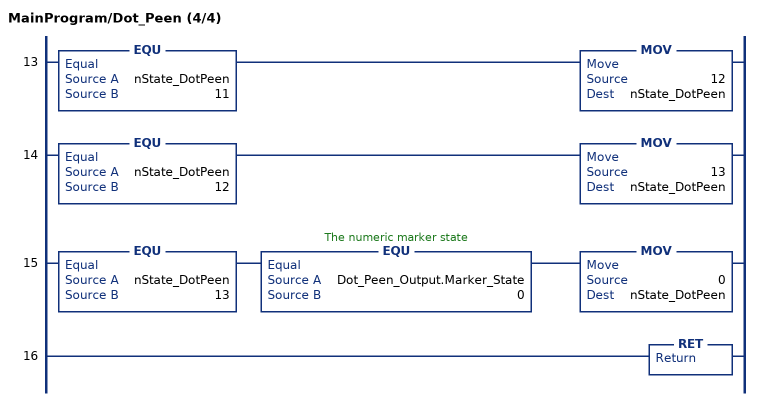
   13: EQU(nState_DotPeen,11)MOV(12,nState_DotPeen);
   14: EQU(nState_DotPeen,12)MOV(13,nState_DotPeen);
   15: EQU(nState_DotPeen,13)EQU(Dot_Peen_Output.Marker_State,0)MOV(0,nState_DotPeen);
   16: RET();
END_ROUTINE

ROUTINE Dot_Peen_AOI   (* ladder *)
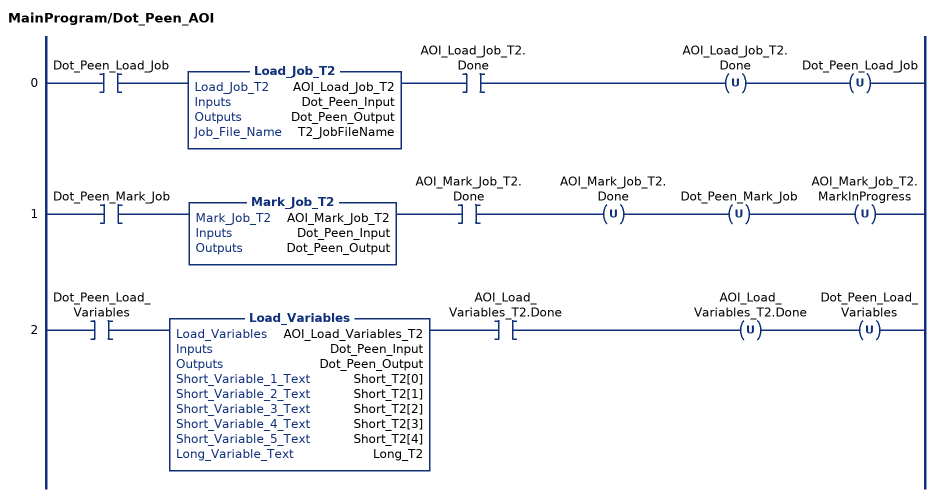
   0: XIC(Dot_Peen_Load_Job)Load_Job_T2(AOI_Load_Job_T2,Dot_Peen_Input,Dot_Peen_Output,T2_JobFileName)XIC(AOI_Load_Job_T2.Done)OTU(AOI_Load_Job_T2.Done)OTU(Dot_Peen_Load_Job);
   1: XIC(Dot_Peen_Mark_Job)Mark_Job_T2(AOI_Mark_Job_T2,Dot_Peen_Input,Dot_Peen_Output)XIC(AOI_Mark_Job_T2.Done)OTU(AOI_Mark_Job_T2.Done)OTU(Dot_Peen_Mark_Job)OTU(AOI_Mark_Job_T2.MarkInProgress);
   2: XIC(Dot_Peen_Load_Variables)Load_Variables(AOI_Load_Variables_T2,Dot_Peen_Input,Dot_Peen_Output,Short_T2[0],Short_T2[1],Short_T2[2],Short_T2[3],Short_T2[4],Long_T2)XIC(AOI_Load_Variables_T2.Done)OTU(AOI_Load_Variables_T2.Done)OTU(Dot_Peen_Load_Variables);
END_ROUTINE

ROUTINE Laser   (* ladder *)
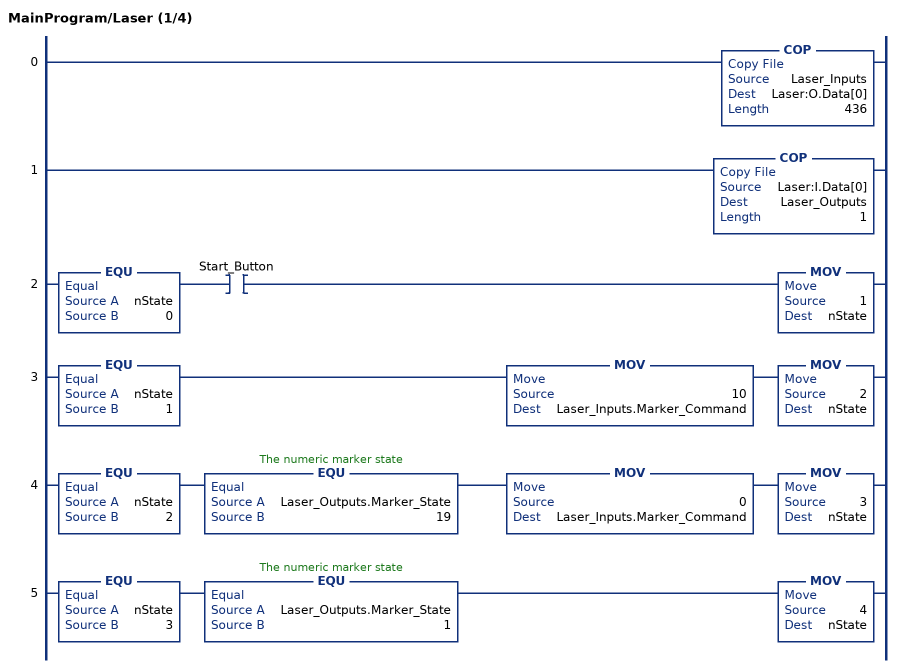
   0: COP(Laser_Inputs,Laser:O.Data[0],436);
   1: COP(Laser:I.Data[0],Laser_Outputs,1);
   2: EQU(nState,0)XIC(Start_Button)MOV(1,nState);
   3: EQU(nState,1)MOV(10,Laser_Inputs.Marker_Command)MOV(2,nState);
   4: EQU(nState,2)EQU(Laser_Outputs.Marker_State,19)MOV(0,Laser_Inputs.Marker_Command)MOV(3,nState);
   5: EQU(nState,3)EQU(Laser_Outputs.Marker_State,1)MOV(4,nState);
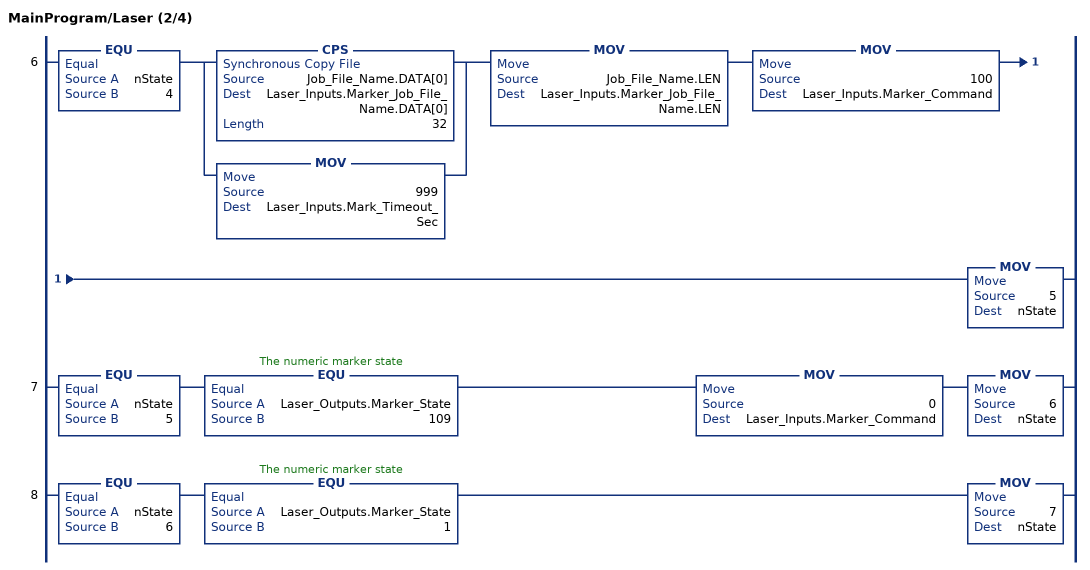
   6: EQU(nState,4)[CPS(Job_File_Name.DATA[0],Laser_Inputs.Marker_Job_File_Name.DATA[0],32) ,MOV(999,Laser_Inputs.Mark_Timeout_Sec) ]MOV(Job_File_Name.LEN,Laser_Inputs.Marker_Job_File_Name.LEN)MOV(100,Laser_Inputs.Marker_Command)MOV(5,nState);
   7: EQU(nState,5)EQU(Laser_Outputs.Marker_State,109)MOV(0,Laser_Inputs.Marker_Command)MOV(6,nState);
   8: EQU(nState,6)EQU(Laser_Outputs.Marker_State,1)MOV(7,nState);
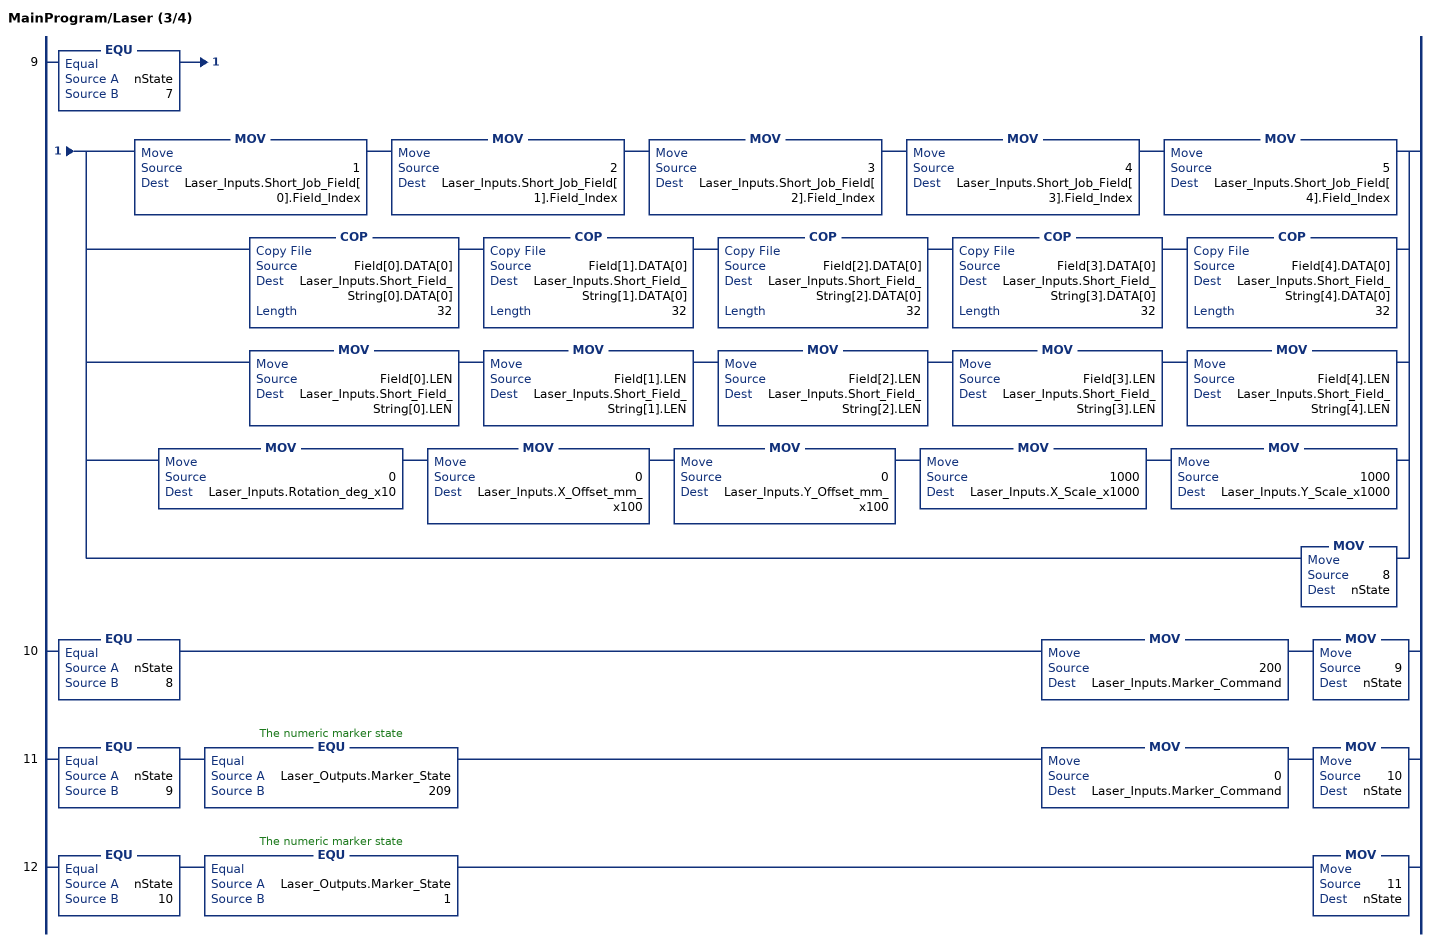
   9: EQU(nState,7)[MOV(1,Laser_Inputs.Short_Job_Field[0].Field_Index) MOV(2,Laser_Inputs.Short_Job_Field[1].Field_Index) MOV(3,Laser_Inputs.Short_Job_Field[2].Field_Index) MOV(4,Laser_Inputs.Short_Job_Field[3].Field_Index) MOV(5,Laser_Inputs.Short_Job_Field[4].Field_Index) ,COP(Field[0].DATA[0],Laser_Inputs.Short_Field_String[0].DATA[0],32) COP(Field[1].DATA[0],Laser_Inputs.Short_Field_String[1].DATA[0],32) COP(Field[2].DATA[0],Laser_Inputs.Short_Field_String[2].DATA[0],32) COP(Field[3].DATA[0],Laser_Inputs.Short_Field_String[3].DATA[0],32) COP(Field[4].DATA[0],Laser_Inputs.Short_Field_String[4].DATA[0],32) ,MOV(Field[0].LEN,Laser_Inputs.Short_Field_String[0].LEN) MOV(Field[1].LEN,Laser_Inputs.Short_Field_String[1].LEN) MOV(Field[2].LEN,Laser_Inputs.Short_Field_String[2].LEN) MOV(Field[3].LEN,Laser_Inputs.Short_Field_String[3].LEN) MOV(Field[4].LEN,Laser_Inputs.Short_Field_String[4].LEN) ,MOV(0,Laser_Inputs.Rotation_deg_x10) MOV(0,Laser_Inputs.X_Offset_mm_x100) MOV(0,Laser_Inputs.Y_Offset_mm_x100) MOV(1000,Laser_Inputs.X_Scale_x1000) MOV(1000,Laser_Inputs.Y_Scale_x1000) ,MOV(8,nState) ];
   10: EQU(nState,8)MOV(200,Laser_Inputs.Marker_Command)MOV(9,nState);
   11: EQU(nState,9)EQU(Laser_Outputs.Marker_State,209)MOV(0,Laser_Inputs.Marker_Command)MOV(10,nState);
   12: EQU(nState,10)EQU(Laser_Outputs.Marker_State,1)MOV(11,nState);
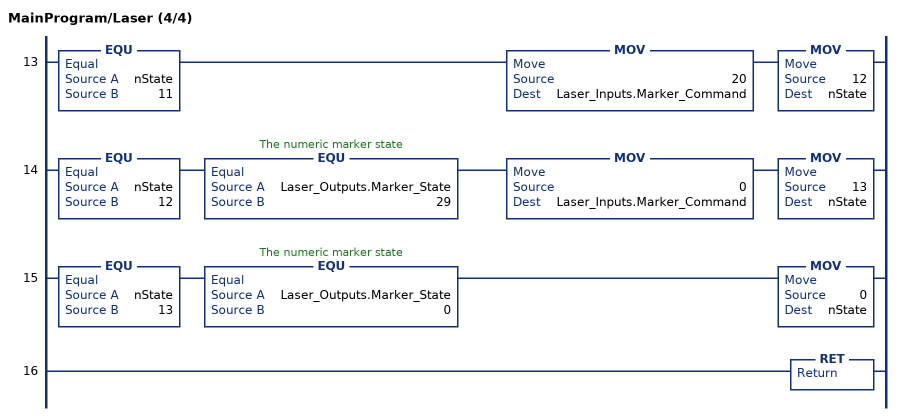
   13: EQU(nState,11)MOV(20,Laser_Inputs.Marker_Command)MOV(12,nState);
   14: EQU(nState,12)EQU(Laser_Outputs.Marker_State,29)MOV(0,Laser_Inputs.Marker_Command)MOV(13,nState);
   15: EQU(nState,13)EQU(Laser_Outputs.Marker_State,0)MOV(0,nState);
   16: RET();
END_ROUTINE

ROUTINE Laser_AOI   (* ladder *)
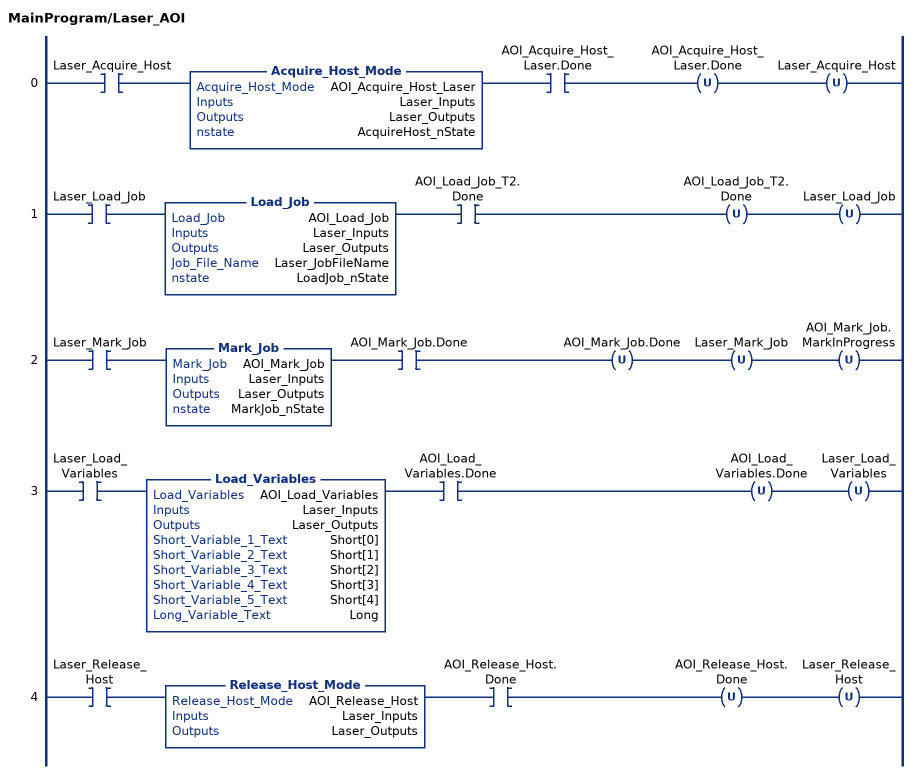
   0: XIC(Laser_Acquire_Host)Acquire_Host_Mode(AOI_Acquire_Host_Laser,Laser_Inputs,Laser_Outputs,AcquireHost_nState)XIC(AOI_Acquire_Host_Laser.Done)OTU(AOI_Acquire_Host_Laser.Done)OTU(Laser_Acquire_Host);
   1: XIC(Laser_Load_Job)Load_Job(AOI_Load_Job,Laser_Inputs,Laser_Outputs,Laser_JobFileName,LoadJob_nState)XIC(AOI_Load_Job_T2.Done)OTU(AOI_Load_Job_T2.Done)OTU(Laser_Load_Job);
   2: XIC(Laser_Mark_Job)Mark_Job(AOI_Mark_Job,Laser_Inputs,Laser_Outputs,MarkJob_nState)XIC(AOI_Mark_Job.Done)OTU(AOI_Mark_Job.Done)OTU(Laser_Mark_Job)OTU(AOI_Mark_Job.MarkInProgress);
   3: XIC(Laser_Load_Variables)Load_Variables(AOI_Load_Variables,Laser_Inputs,Laser_Outputs,Short[0],Short[1],Short[2],Short[3],Short[4],Long)XIC(AOI_Load_Variables.Done)OTU(AOI_Load_Variables.Done)OTU(Laser_Load_Variables);
   4: XIC(Laser_Release_Host)Release_Host_Mode(AOI_Release_Host,Laser_Inputs,Laser_Outputs)XIC(AOI_Release_Host.Done)OTU(AOI_Release_Host.Done)OTU(Laser_Release_Host);
END_ROUTINE

ROUTINE MainRoutine   (* ladder *)
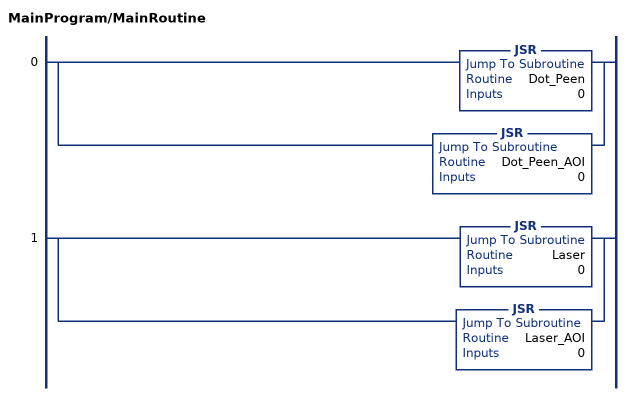
   0: [JSR(Dot_Peen,0) ,JSR(Dot_Peen_AOI,0) ];
   1: [JSR(Laser,0) ,JSR(Laser_AOI,0) ];
END_ROUTINE
END_PROGRAM
